SYSTEM DASDAass2 (* System Configuration *)
  (* Standard: 61499-1 *)
  (* Version 0.4, 2009-03-05, JHC, Holobloc Inc., Deleted Application. *)
  (* Version 0.3, 2003-12-05, JHC, Rockwell Automation, Renamed from NEWSYSTEM. *)
  (* Version 0.2, 2002-11-05, JHC, Rockwell Automation, Fixed missing (empty) FBD in Application. *)
  (* Version 0.1, 2002-01-17, JHC, Rockwell Automation, Minor cleanup *)
  (* Version 0.0, 2000-05-27, JHC, Rockwell Automation *)
  DEVICE VIEW_LAYER : FRAME_DEVICE(BOUNDS := [200,0,250,200])
    RESOURCE VIEW_RES : VIEW_PANEL(DIA := 25, SIZE := [10,8], VERTICAL := 0)
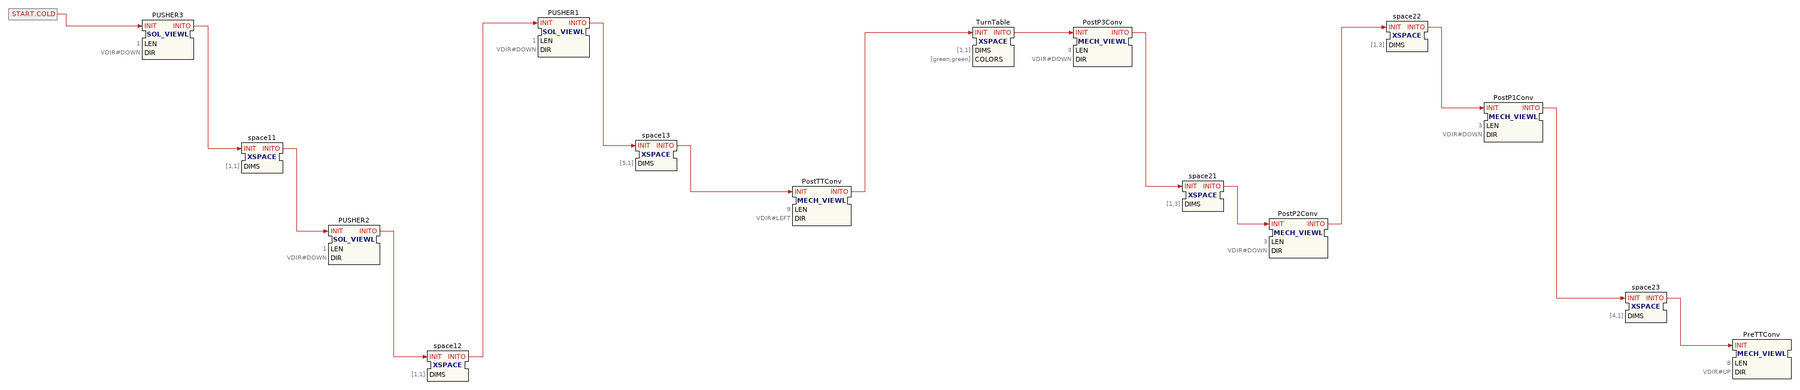
      FBS
        PUSHER3 : SOL_VIEWL(LEN := 1, DIR := VDIR#DOWN);
        space11 : XSPACE(DIMS := [1,1]);
        PUSHER2 : SOL_VIEWL(LEN := 1, DIR := VDIR#DOWN);
        space12 : XSPACE(DIMS := [1,1]);
        PUSHER1 : SOL_VIEWL(LEN := 1, DIR := VDIR#DOWN);
        space13 : XSPACE(DIMS := [5,1]);
        PostTTConv : MECH_VIEWL(LEN := 9, DIR := VDIR#LEFT); (* Supply transfer mechanism *)
        TurnTable : XSPACE(DIMS := [1,1], COLORS := [green,green]);
        PostP3Conv : MECH_VIEWL(LEN := 3, DIR := VDIR#DOWN); (* Supply transfer mechanism *)
        space21 : XSPACE(DIMS := [1,3]);
        PostP2Conv : MECH_VIEWL(LEN := 3, DIR := VDIR#DOWN); (* Supply transfer mechanism *)
        space22 : XSPACE(DIMS := [1,3]);
        PostP1Conv : MECH_VIEWL(LEN := 3, DIR := VDIR#DOWN); (* Supply transfer mechanism *)
        space23 : XSPACE(DIMS := [4,1]);
        PreTTConv : MECH_VIEWL(LEN := 8, DIR := VDIR#UP); (* Supply transfer mechanism *)
      END_FBS
      EVENT_CONNECTIONS
        START.COLD TO PUSHER3.INIT;
        PUSHER3.INITO TO space11.INIT;
        space11.INITO TO PUSHER2.INIT;
        PUSHER2.INITO TO space12.INIT;
        space12.INITO TO PUSHER1.INIT;
        PUSHER1.INITO TO space13.INIT;
        space13.INITO TO PostTTConv.INIT;
        TurnTable.INITO TO PostP3Conv.INIT;
        PostP3Conv.INITO TO space21.INIT;
        space21.INITO TO PostP2Conv.INIT;
        PostP2Conv.INITO TO space22.INIT;
        space22.INITO TO PostP1Conv.INIT;
        PostP1Conv.INITO TO space23.INIT;
        space23.INITO TO PreTTConv.INIT;
        PostTTConv.INITO TO TurnTable.INIT;
      END_CONNECTIONS
    END_RESOURCE
  END_DEVICE
  DEVICE HMI_LAYER : FRAME_DEVICE(BOUNDS := [0,0,200,200])
    RESOURCE HMI_1 : PANEL_RESOURCE(COLS := 1)
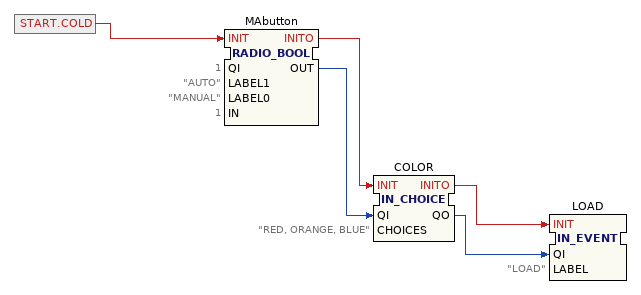
      FBS
        MAbutton : RADIO_BOOL(QI := 1, LABEL1 := "AUTO", LABEL0 := "MANUAL", IN := 1);
        LOAD : IN_EVENT(LABEL := "LOAD");
        COLOR : IN_CHOICE(CHOICES := "RED, ORANGE, BLUE");
      END_FBS
      EVENT_CONNECTIONS
        START.COLD TO MAbutton.INIT;
        COLOR.INITO TO LOAD.INIT;
        MAbutton.INITO TO COLOR.INIT;
      END_CONNECTIONS
      DATA_CONNECTIONS
        COLOR.QO TO LOAD.QI;
        MAbutton.OUT TO COLOR.QI;
      END_CONNECTIONS
    END_RESOURCE
  END_DEVICE
END_SYSTEM
